INTERFACE EventLogger

PROPERTY PUBLIC level : EventLevel
GET
END_GET
SET
END_SET
END_PROPERTY

METHOD run
VAR_INPUT
  act_time: TIMESTRUCT;
END_VAR
END_METHOD

METHOD PUBLIC submit_event_message
VAR_INPUT
  ev: EventMessage;
END_VAR
END_METHOD

END_INTERFACE

(* stored: Version 1.1.0.1, ProductVersion 3.1.4024.9
   Itf EventLogger: Id {ed02ee8e-c48d-425b-b1ba-db2fe412fd83}
   Property level: Id {730b9c5a-0551-4f93-88c2-7713947006a0}
   Get Get: Id {841b1b39-fa57-4400-953f-380c944e25b0}
   Set Set: Id {969b46fd-305f-40c3-b3af-abdb26bc71cc}
   Method run: Id {aef2808e-85b7-4075-9c20-5b0b7eee7fcc}
   Method submit_event_message: Id {f84ec892-41c2-4113-b29d-b2de8225110c} *)
